Fanuc KAREL source: kt00216.KL

-- PROVISIONAL review KL for V1013-1; original PC SHA256 a13283e17f6e9a18a96bfe2b02b67c7f1c48f47b3a6b60d1d9866b4eb72cafce
-- Incomplete behavior may be omitted. Consult companion uncertainty JSON. Do not deploy.
PROGRAM KT00216
%NOLOCKGROUP
VAR
  OUT : INTEGER
-- UNRESOLVED_DECL Y1 type=002018
-- UNRESOLVED_DECL H2 type=002017
BEGIN
  -- UNRESOLVED_PC offsets 5-19; opcodes 2E,22,9D,33,B2
  -- UNRESOLVED_PC offsets 24-38; opcodes 2E,22,9D,33,B4
  -- UNRESOLVED_PC offsets 43-68; opcodes 22,9D,33,B1,22,9D,33,B3,46,23
  -- UNRESOLVED_PC offsets 73-77; opcodes 7F
END KT00216
